FUNCTION_BLOCK ROBOT6TESTFB (* JADE WORKER *)
  (* Standard: 61499-1 *)
  (* Version 1.0, 2014-04-22, Ahmed, Fraunhofer IGD *)
  (* Compiler header: package fb.rt; *)
  (* Compiler Java Sun JDK 1.5.0 *)
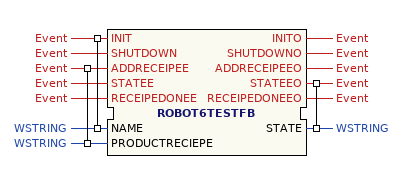
  EVENT_INPUT
    INIT WITH NAME; (* Normal Execution Request *)
    SHUTDOWN;
    ADDRECEIPEE WITH PRODUCTRECIEPE; (* Normal Execution Request *)
    STATEE;
    RECEIPEDONEE;
  END_EVENT
  EVENT_OUTPUT
    INITO; (* Execution Confirmation *)
    SHUTDOWNO;
    ADDRECEIPEEO; (* Execution Confirmation *)
    STATEEO WITH STATE;
    RECEIPEDONEEO;
  END_EVENT
  VAR_INPUT
    NAME : WSTRING;
    PRODUCTRECIEPE : WSTRING;
  END_VAR
  VAR_OUTPUT
    STATE : WSTRING;
  END_VAR
END_FUNCTION_BLOCK
